// Automatisch erzeugter Code: NICHT EDITIEREN
FUNCTION CheckLRangeSigned : LINT
VAR_INPUT
	value, lower, upper: LINT;
END_VAR

// Automatisch erzeugter Code: Es handelt sich hierbei um einen Implementierungsvorschlag.
{noflow}
IF (value < lower) THEN
	CheckLRangeSigned := lower;
ELSIF(value > upper) THEN
	CheckLRangeSigned := upper;
ELSE
	CheckLRangeSigned := value;
END_IF

{flow}

END_FUNCTION

(* stored: Version 1.1.0.1, ProductVersion 3.1.4024.10
   POU CheckLRangeSigned: Id {60a6e0c5-6492-4ab1-b34f-2910c28e13e2}, SpecialFunc CheckLRangeSigned *)
